ABB RAPID module: Wizard.modx

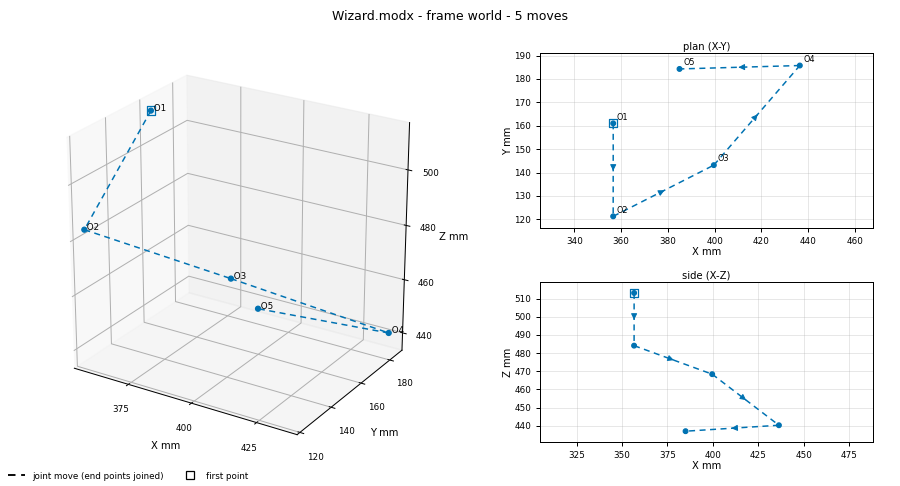
[picture p0: tool path of Wizard.modx in frame world, 5 of 5 moves have a stored position in this frame; points joined in program order, loops and branches not executed]
MODULE Wizard
PERS robtarget O1:=[[356.637451171875, 161.037048339844, 513.128356933594], [0.0388496816158295, -0.776131391525269, -0.358248889446259, -0.517463564872742], [0, 1, 0, 1], [9000000000, 9000000000, 9000000000, 9000000000, 9000000000, 9000000000]];
PERS robtarget O2:=[[356.619445800781, 121.282089233398, 484.093872070313], [0.00313940364867449, -0.806082367897034, -0.327470064163208, -0.492934823036194], [0, 1, 0, 1], [9000000000, 9000000000, 9000000000, 9000000000, 9000000000, 9000000000]];
PERS robtarget O3:=[[399.640594482422, 143.169784545898, 468.373107910156], [0.00769960461184382, 0.794183015823364, 0.382436096668243, 0.472182840108871], [0, 1, 0, 1], [9000000000, 9000000000, 9000000000, 9000000000, 9000000000, 9000000000]];
PERS robtarget O4:=[[436.398681640625, 185.750854492188, 440.245086669922], [0.083333015441895, -0.836603939533234, -0.298512071371078, -0.451707899570465], [0, 1, 0, 1], [9000000000, 9000000000, 9000000000, 9000000000, 9000000000, 9000000000]];
PERS robtarget O5:=[[384.975860595703, 184.290008544922, 436.962097167969], [0.130016103386879, -0.904695689678192, -0.099378101527691, -0.393377006053925], [0, 1, 0, 1], [9000000000, 9000000000, 9000000000, 9000000000, 9000000000, 9000000000]];
	PROC main()
MoveJ O1, v1000, fine, tool0;
MoveJ O2, v1000, fine, tool0;
MoveJ O3, v1000, fine, tool0;
MoveJ O4, v1000, fine, tool0;
MoveJ O5, v1000, fine, tool0;
	ENDPROC
ENDMODULE
